// TIA Portal project "P1_Ejercicio1" (V15.1)

(* hardware
DEVICE "S7-1200 station_1"  S7-1200 Station
   slot 0: "Rack_0"  S7-1200 Rack  Rack  V1.0
   slot 1: "PLC_1"  CPU 1215C AC/DC/Rly  6ES7 215-1BG40-0XB0  V4.2
DEVICE "HMI_1"  KTP900 Basic PN Portrait
   slot 0: "HMI_1"  KTP900 Basic PN Portrait  6AV2 123-2JB03-0AX0  15.1.0.0
   slot 1: "HMI_RT_1"  KTP900 Basic PN Portrait  6AV2 123-2JB03-0AX0  15.1.0.0
   slot 5: "HMI_1.IE_CP_1"  PROFINET Interface  15.0.1.0
      slot 1: "Interfaz PROFINET_1"  PROFINET Interface
         slot 1: "Port_1"  Port
*)

// ===== PLC "PLC_1"  CPU 1215C AC/DC/Rly =====

VAR_GLOBAL   // PLC tag table "Tabla de variables estándar"
   "Interruptor on/off" AT %M0.0 : Bool;
   "Palanca de giro positivo motor" AT %M0.1 : Bool;
   "Palanca de giro negativo motor" AT %M0.2 : Bool;
   "Lámpara funcionamiento" AT %M10.0 : Bool;
   "Lámpara sentido positivo giro" AT %M10.1 : Bool;
   "Lámpara sentido negativo giro" AT %M10.2 : Bool;
   "Contactor giro positivo motor" AT %M10.3 : Bool;
   "Contactor giro negativo motor" AT %M10.4 : Bool;
   "Sensor temperatura" AT %M0.3 : Bool;
   "Piloto panel de mando" AT %M10.5 : Bool;
END_VAR

ORGANIZATION_BLOCK "Main"   // OB1, LAD, ProgramCycle
TITLE = "Main Program Sweep (Cycle)"
{ S7_Optimized_Access := 'TRUE' }
VERSION : 0.1
   VAR_INPUT
      Initial_Call : Bool;   // Initial call of this OB
      Remanence : Bool;   // =True, if remanent data are available
   END_VAR
   VAR_TEMP   // added for the SCL form of the ladder/FBD networks
      _w1 : Bool;
      _w2 : Bool;
   END_VAR
BEGIN

REGION Network 1
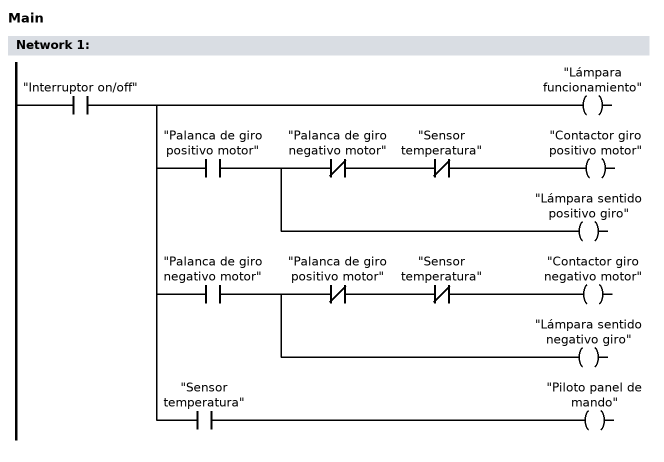
   RUNG wire#powerrail
      Contact( "Interruptor on/off" )
      wire#w1
      Coil( "Lámpara funcionamiento" )
   END_RUNG
   RUNG wire#w1
      Contact( "Palanca de giro positivo motor" )
      wire#w2
      I_Contact( "Palanca de giro negativo motor" )
      I_Contact( "Sensor temperatura" )
      Coil( "Contactor giro positivo motor" )
   END_RUNG
   RUNG wire#w2
      Coil( "Lámpara sentido positivo giro" )
   END_RUNG
   RUNG wire#w1
      Contact( "Palanca de giro negativo motor" )
      wire#w3
      I_Contact( "Palanca de giro positivo motor" )
      I_Contact( "Sensor temperatura" )
      Coil( "Contactor giro negativo motor" )
   END_RUNG
   RUNG wire#w3
      Coil( "Lámpara sentido negativo giro" )
   END_RUNG
   RUNG wire#w1
      Contact( "Sensor temperatura" )
      Coil( "Piloto panel de mando" )
   END_RUNG
   // the same network as SCL:
   "Lámpara funcionamiento" := "Interruptor on/off";
   #_w1 := "Interruptor on/off" AND "Palanca de giro positivo motor";
   "Contactor giro positivo motor" := #_w1 AND NOT "Palanca de giro negativo motor" AND NOT "Sensor temperatura";
   "Lámpara sentido positivo giro" := #_w1;
   #_w2 := "Interruptor on/off" AND "Palanca de giro negativo motor";
   "Contactor giro negativo motor" := #_w2 AND NOT "Palanca de giro positivo motor" AND NOT "Sensor temperatura";
   "Lámpara sentido negativo giro" := #_w2;
   "Piloto panel de mando" := "Interruptor on/off" AND "Sensor temperatura";
END_REGION
END_ORGANIZATION_BLOCK

(* ===== HMI "HMI_RT_1" =====
system functions are stored by id; their names below are inferred from use
connection "HMI_Conexión_1": ETHERNET, SMART_S7_1200_OMS

HMI tags "Tabla de variables estándar"
   "Número_imagen_variable" : UInt, internal
   "Interruptor on/off" : Bool = PLC "Interruptor on/off" AT %M0.0, 1 s
   "Lámpara funcionamiento" : Bool = PLC "Lámpara funcionamiento" AT %M10.0, 1 s
   "Lámpara sentido positivo giro" : Bool = PLC "Lámpara sentido positivo giro" AT %M10.1, 1 s
   "Palanca de giro positivo motor" : Bool = PLC "Palanca de giro positivo motor" AT %M0.1, 1 s
   "Palanca de giro negativo motor" : Bool = PLC "Palanca de giro negativo motor" AT %M0.2, 1 s
   "Lámpara sentido negativo giro" : Bool = PLC "Lámpara sentido negativo giro" AT %M10.2, 1 s
   "Piloto panel de mando" : Bool = PLC "Piloto panel de mando" AT %M10.5, 1 s

text list "Nombre_imagen_lista_texto": 1 'Imagen raíz'

Template "Plantilla_1" 480x800
   Button "Imagen inicial" at 439,57 size 39x55; TextOff 'Imagen inicial'; PictureOff "NavigateHome_KTP900_Basic_PN_Portrait_TR"; PictureOn "NavigateHome_KTP900_Basic_PN_Portrait_TR"
      on Release: ActivateScreen("Imagen raíz", 0)
   Button "Avisos" at 439,171 size 39x55; TextOff 'Avisos'; PictureOff "AlarmDisplay_KTP900_Basic_PN_Portrait_TR"; PictureOn "AlarmDisplay_KTP900_Basic_PN_Portrait_TR"
      on Release: function_ef3f5d25("Ventana de avisos_no_acusado", -1)
   Button "Template_Button" at 439,286 size 39x55; TextOff 'Text'
   Button "Template_Button_1" at 439,400 size 39x55; TextOff 'Text'
   Button "Template_Button_2" at 439,514 size 39x55; TextOff 'Text'
   Button "Template_Button_3" at 439,629 size 39x55; TextOff 'Text'
   Button "Salir" at 439,743 size 39x55; TextOff 'Salir'; PictureOff "ExitRuntime_KTP900_Basic_PN_Portrait_TR"; PictureOn "ExitRuntime_KTP900_Basic_PN_Portrait_TR"
      on Release: StopRuntime(0)
   SymbolicIOField "Imagen_campo_ES_simbólico" at 102,10 size 271x36; TextOff '0'; TextOn '1'; TextList "Nombre_imagen_lista_texto"
      ProcessValue <- "Número_imagen_variable"
      on Change: ActivateScreenByNumber("Número_imagen_variable", 0)
   DateTimeField "HmiScreenItemData" at 375,28 size 105x28
   DateTimeField "HmiScreenItemData_1" at 375,0 size 105x28
   GraphicView "Logotipo" at 0,0 size 100x56; Picture "Logotipo de HMI_1"

screen "Imagen raíz" 480x800, template "Plantilla_1"
   on GenerateScreen: SetTag("Número_imagen_variable", 1)
   Switch "Interruptor_1" at 20,102 size 130x45; CaptionText 'Switch'; TextOff 'OFF'; TextOn 'ON'
      ProcessValue <- "Interruptor on/off"
   TextField "Campo de texto_1" at 20,76 size 130x20; Text 'Interruptor ON/OFF'
   Circle "Círculo_1" at 325,102 size 48x48
      Appearance <- "Lámpara funcionamiento"
   TextField "Campo de texto_2" at 263,82 size 164x20; Text 'Lámpara funcionamiento'
   Switch "Interruptor_2" at 96,222 size 92x31; TextOn 'ON'; CaptionText 'Switch'; TextOff 'OFF'
      ProcessValue <- "Palanca de giro positivo motor"
   Switch "Interruptor_3" at 96,315 size 92x31; TextOn 'ON'; CaptionText 'Switch'; TextOff 'OFF'
      ProcessValue <- "Palanca de giro negativo motor"
   Circle "Círculo_2" at 325,214 size 48x48
      Appearance <- "Lámpara sentido positivo giro"
   Circle "Círculo_3" at 325,305 size 48x48
      Appearance <- "Lámpara sentido negativo giro"
   TextField "Campo de texto_3" at 71,194 size 159x20; Text 'Palanca de giro positivo'
   TextField "Campo de texto_4" at 71,285 size 165x20; Text 'Palanca de giro negativo'
   TextField "Campo de texto_5" at 282,194 size 145x20; Text 'Lámpara giro positivo'
   TextField "Campo de texto_6" at 284,285 size 151x20; Text 'Lámpara giro negativo'
   Rectangle "Rectángulo_1" at 277,419 size 96x48
      Appearance <- "Piloto panel de mando"
   TextField "Campo de texto_7" at 242,392 size 171x21; Text 'Piloto de panel de mando'
*)